// TIA Portal V20 export
DATA_BLOCK "LDrvSafe_SinaTlg701Status_DB_DR31"   // DB386
FAMILY : LDrvSafe
VERSION : 2.0
// stored: InstanceOfName LDrvSafe_SinaTlg701Status, InstanceOfType FB, Namespace Unit1
"LDrvSafe_SinaTlg701Status"
   // VAR_INPUT
   //    enable : Bool := FALSE;
   //    hardwareId : HW_IO := 0;
   // END_VAR
   // VAR_OUTPUT
   //    valid { ExternalWritable := 'False'} : Bool := FALSE;
   //    busy { ExternalWritable := 'False'} : Bool := FALSE;
   //    error { ExternalWritable := 'False'} : Bool := FALSE;
   //    status { ExternalWritable := 'False'} : Word := 16#7000;
   //    safetyFaultActive { ExternalWritable := 'False'} : Bool := FALSE;
   //    safetyMessageActive { ExternalWritable := 'False'} : Bool := FALSE;
   //    STOactive { ExternalWritable := 'False'} : Bool := FALSE;
   //    SS1active { ExternalWritable := 'False'} : Bool := FALSE;
   //    SS1Eactive { ExternalWritable := 'False'} : Bool := FALSE;
   //    SS2active { ExternalWritable := 'False'} : Bool := FALSE;
   //    SS2Eactive { ExternalWritable := 'False'} : Bool := FALSE;
   //    SS2ESRactive { ExternalWritable := 'False'} : Bool := FALSE;
   //    SOSselected { ExternalWritable := 'False'} : Bool := FALSE;
   //    SOSactive { ExternalWritable := 'False'} : Bool := FALSE;
   //    SLSselected { ExternalWritable := 'False'} : Bool := FALSE;
   //    SLSactive { ExternalWritable := 'False'} : Bool := FALSE;
   //    SLSbit0Active { ExternalWritable := 'False'} : Bool := FALSE;
   //    SLSbit1Active { ExternalWritable := 'False'} : Bool := FALSE;
   //    SLPrangeSelected { ExternalWritable := 'False'} : Bool := FALSE;
   //    SLPselectedAndUserAgreement { ExternalWritable := 'False'} : Bool := FALSE;
   //    referencePositionRequired { ExternalWritable := 'False'} : Bool := FALSE;
   //    referencePositionValid { ExternalWritable := 'False'} : Bool := FALSE;
   //    SLAactive { ExternalWritable := 'False'} : Bool := FALSE;
   //    SDIpositiveSelected { ExternalWritable := 'False'} : Bool := FALSE;
   //    SDInegativeSelected { ExternalWritable := 'False'} : Bool := FALSE;
   //    SDIpositive { ExternalWritable := 'False'} : Bool := FALSE;
   //    SDInegative { ExternalWritable := 'False'} : Bool := FALSE;
   //    ESRretractRequested { ExternalWritable := 'False'} : Bool := FALSE;
   //    brakeTestSelected { ExternalWritable := 'False'} : Bool := FALSE;
   //    setpointInput { ExternalWritable := 'False'} : Bool := FALSE;
   //    activeBrake { ExternalWritable := 'False'} : Bool := FALSE;
   //    brakeTestActive { ExternalWritable := 'False'} : Bool := FALSE;
   //    brakeTestResult { ExternalWritable := 'False'} : Bool := FALSE;
   //    brakeTestCompleted { ExternalWritable := 'False'} : Bool := FALSE;
   //    externalBrakeRequest { ExternalWritable := 'False'} : Bool := FALSE;
   //    currentLoadSign { ExternalWritable := 'False'} : Bool := FALSE;
   //    acceptanceTestSLPselected { ExternalWritable := 'False'} : Bool := FALSE;
   //    acceptanceTestModeSelected { ExternalWritable := 'False'} : Bool := FALSE;
   //    SLSlimit { ExternalWritable := 'False'} : DWord := 16#0000_0000;
   // END_VAR
   // VAR
   //    statEnableOld { ExternalVisible := 'False'; ExternalWritable := 'False'} : Bool := FALSE;
   //    statValid { ExternalVisible := 'False'; ExternalWritable := 'False'} : Bool := FALSE;
   //    statBusy { ExternalVisible := 'False'; ExternalWritable := 'False'} : Bool := FALSE;
   //    statError { ExternalVisible := 'False'; ExternalWritable := 'False'} : Bool := FALSE;
   //    statErrorRead { ExternalVisible := 'False'; ExternalWritable := 'False'} : Bool := FALSE;
   //    statStatus { ExternalVisible := 'False'; ExternalWritable := 'False'} : Word := 16#7000;
   //    statStatusRead { ExternalVisible := 'False'; ExternalWritable := 'False'} : DWord := 16#0000_0000;
   //    statFBState { ExternalVisible := 'False'; ExternalWritable := 'False'} : DInt := 0;
   //    statDisablingCompleted { ExternalVisible := 'False'; ExternalWritable := 'False'} : Bool := FALSE;
   //    statRecvBuf { ExternalVisible := 'False'; ExternalWritable := 'False'} : "LDrvSafe_typeSinaTlg701Status";
   //    instReadTlg701 { ExternalVisible := 'False'; ExternalWritable := 'False'} : GETIO_PART;
   // END_VAR
BEGIN
   statRecvBuf.S_ZSW1B.SLAactive := FALSE;
   statRecvBuf.S_ZSW1B.SLSbit0Active := FALSE;
   statRecvBuf.S_ZSW1B.SLSbit1Active := FALSE;
   statRecvBuf.S_ZSW1B.reserved := FALSE;
   statRecvBuf.S_ZSW1B.SDIpositiveSelected := FALSE;
   statRecvBuf.S_ZSW1B.SDInegativeSelected := FALSE;
   statRecvBuf.S_ZSW1B.ESRretractRequested := FALSE;
   statRecvBuf.S_ZSW1B.safetyMessageActive := FALSE;
   statRecvBuf.S_ZSW1B.STOactive := FALSE;
   statRecvBuf.S_ZSW1B.SS1active := FALSE;
   statRecvBuf.S_ZSW1B.SS2active := FALSE;
   statRecvBuf.S_ZSW1B.SOSactive := FALSE;
   statRecvBuf.S_ZSW1B.SLSactive := FALSE;
   statRecvBuf.S_ZSW1B.SOSselected := FALSE;
   statRecvBuf.S_ZSW1B.SLSselected := FALSE;
   statRecvBuf.S_ZSW1B.safetyFaultActive := FALSE;
   statRecvBuf.S_ZSW2B.SDIpositive := FALSE;
   statRecvBuf.S_ZSW2B.SDInegative := FALSE;
   statRecvBuf.S_ZSW2B.reserved5 := FALSE;
   statRecvBuf.S_ZSW2B.reserved6 := FALSE;
   statRecvBuf.S_ZSW2B.reserved7 := FALSE;
   statRecvBuf.S_ZSW2B.reserved8 := FALSE;
   statRecvBuf.S_ZSW2B.referencePositionRequired := FALSE;
   statRecvBuf.S_ZSW2B.referencePositionValid := FALSE;
   statRecvBuf.S_ZSW2B.reserved0 := FALSE;
   statRecvBuf.S_ZSW2B.reserved1 := FALSE;
   statRecvBuf.S_ZSW2B.reserved2 := FALSE;
   statRecvBuf.S_ZSW2B.SS1Eactive := FALSE;
   statRecvBuf.S_ZSW2B.SLPrangeSelected := FALSE;
   statRecvBuf.S_ZSW2B.reserved3 := FALSE;
   statRecvBuf.S_ZSW2B.reserved4 := FALSE;
   statRecvBuf.S_ZSW2B.SLPselectedAndUserAgreement := FALSE;
   statRecvBuf.SLSlimit := 16#0000_0000;
   statRecvBuf.S_ZSW3B.reserved0 := FALSE;
   statRecvBuf.S_ZSW3B.reserved1 := FALSE;
   statRecvBuf.S_ZSW3B.reserved2 := FALSE;
   statRecvBuf.S_ZSW3B.SS2Eactive := FALSE;
   statRecvBuf.S_ZSW3B.SS2ESRactive := FALSE;
   statRecvBuf.S_ZSW3B.reserved3 := FALSE;
   statRecvBuf.S_ZSW3B.acceptanceTestSLPselected := FALSE;
   statRecvBuf.S_ZSW3B.acceptanceTestModeSelected := FALSE;
   statRecvBuf.S_ZSW3B.brakeTest := FALSE;
   statRecvBuf.S_ZSW3B.setpointInput := FALSE;
   statRecvBuf.S_ZSW3B.activeBrake := FALSE;
   statRecvBuf.S_ZSW3B.brakeTestActive := FALSE;
   statRecvBuf.S_ZSW3B.brakeTestResult := FALSE;
   statRecvBuf.S_ZSW3B.brakeTestCompleted := FALSE;
   statRecvBuf.S_ZSW3B.externalBrakeRequest := FALSE;
   statRecvBuf.S_ZSW3B.currentLoadSign := FALSE;
   instReadTlg701.ID := 0;
   instReadTlg701.OFFSET := 0;
   instReadTlg701.LEN := 0;
   instReadTlg701.STATUS := 16#0000_0000;
   instReadTlg701.ERROR := FALSE;
END_DATA_BLOCK
